INTERFACE I_State

METHOD Cancel : BOOL
VAR_INPUT
END_VAR
END_METHOD

METHOD Card_Ejected : BOOL
VAR_INPUT
END_VAR
END_METHOD

METHOD Card_Inserted : BOOL
VAR_INPUT
END_VAR
END_METHOD

PROPERTY Description : E_StateDescription
GET
END_GET
END_PROPERTY

METHOD Failure : BOOL
VAR_INPUT
END_VAR
END_METHOD

METHOD Op : BOOL
VAR_INPUT
END_VAR
END_METHOD

METHOD Service : BOOL
VAR_INPUT
END_VAR
END_METHOD

METHOD SystemTest_OK : BOOL
VAR_INPUT
END_VAR
END_METHOD

METHOD Turn_Off : BOOL
VAR_INPUT
END_VAR
END_METHOD

METHOD Turn_On : BOOL
VAR_INPUT
END_VAR
END_METHOD

END_INTERFACE

(* stored: Version 1.1.0.1, ProductVersion 3.1.4024.12
   Itf I_State: Id {a1c71530-fa84-0bb0-3283-cd1f622ad3a9}
   Method Cancel: Id {f6bb5175-37f0-0176-291d-a4d7620ac1d5}
   Method Card_Ejected: Id {2a05fd73-eee8-07e4-06be-b024194c550e}
   Method Card_Inserted: Id {b2d4e578-f718-0e93-0b18-a80f84b9017f}
   Property Description: Id {44bc2097-a004-0b24-1095-c71e11eeaf2b}
   Get Get: Id {c2a9615a-f216-0b01-309d-59e63ba0df67}
   Method Failure: Id {21c6a420-876b-0f5b-241e-27ee63e097b3}
   Method Op: Id {3a5100e4-d2c3-0577-3937-c05a43814309}
   Method Service: Id {94cbab84-9e89-079e-1c59-18b9122a858e}
   Method SystemTest_OK: Id {66832ca6-a287-098d-31cb-ca7c9c991d32}
   Method Turn_Off: Id {57f5bb9a-c5f8-0ce1-0804-28a0bdf1434e}
   Method Turn_On: Id {6119d6b8-41b5-08be-17d1-44b4e801e015} *)
